ABB RobotStudio station: myGofa.rsstn

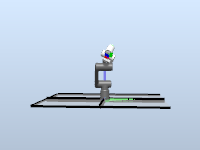
Station myGofa (saved by RobotStudio 21.2.9526.0)
Controller CRB15000_5_95
  mechanical unit ROB_1: CRB15000_5_95__01, 6 joints, base frame (0, 0, 0) mm
Layout (positions relative to the parent item):
  - CRB15000_5_95__01 [mechanism, from Robots\CRB15000_5_95__01.rslib] at (0, 0, 0) mm; joint values [0.1219, 0.8471, -0.9975, -0.4613, 0.7267, 0.2435] (rad or m)
